INTERFACE IEcTask EXTENDS ITask

PROPERTY NetID : amsnetid
GET
END_GET
SET
END_SET
END_PROPERTY

END_INTERFACE

(* stored: Version 1.1.0.1, ProductVersion 3.1.4024.11
   Itf IEcTask: Id {4f801423-2ae2-40da-928f-fc137535ccfd}
   Property NetID: Id {0875c1fc-45fd-4572-a34d-d8ceac62a048}
   Get Get: Id {05810287-a198-42bf-bf95-9ca4aafca301}
   Set Set: Id {639d7282-a26a-45ea-a621-7cfae3eb197c} *)
